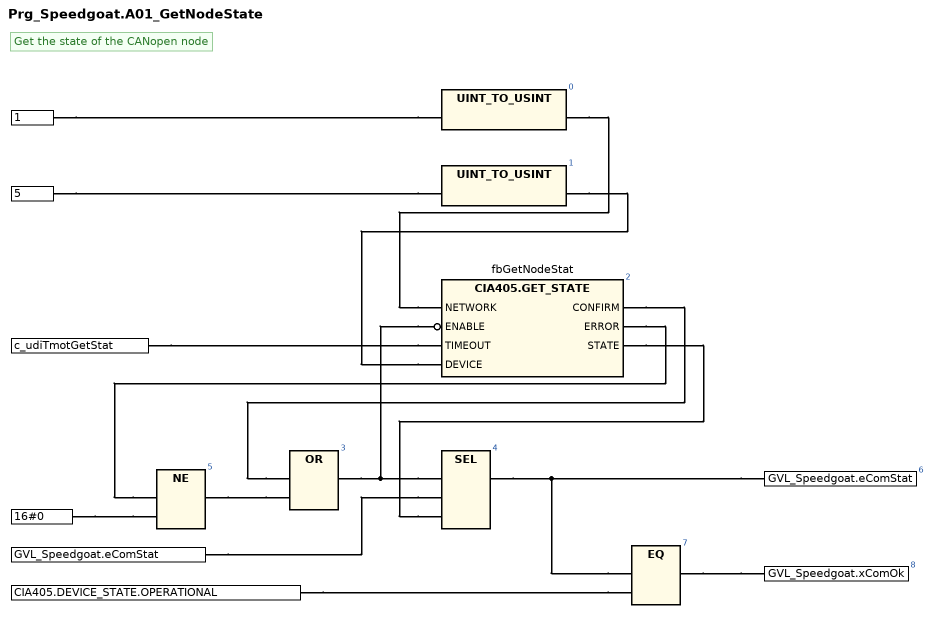
// Get the state of the CANopen node
fbGetNodeStat(
    NETWORK := UINT_TO_USINT(1),
    ENABLE := NOT _w1,
    TIMEOUT := c_udiTmotGetStat,
    DEVICE := UINT_TO_USINT(5)); // CIA405.GET_STATE
_w1 := fbGetNodeStat.CONFIRM OR _w2;
_w3 := SEL(_w1, GVL_Speedgoat.eComStat, fbGetNodeStat.STATE);
_w2 := fbGetNodeStat.ERROR <> 16#0;
GVL_Speedgoat.eComStat := _w3;
GVL_Speedgoat.xComOk := _w3 = CIA405.DEVICE_STATE.OPERATIONAL;
END_ACTION

END_PROGRAM

// HMISAC/Application/AlarmManager
PROGRAM AlarmManager
VAR
END_VAR

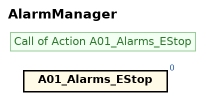
// Call of Action A01_Alarms_EStop
A01_Alarms_EStop();

ACTION A06_Alarms_LXM32i_Node11:
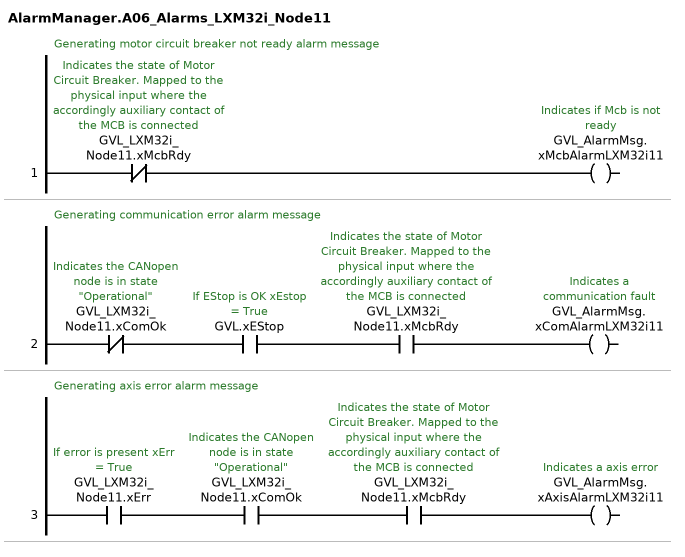
// NETWORK 1
// Generating motor circuit breaker not ready alarm message
//   GVL_LXM32i_Node11.xMcbRdy: Indicates the state of Motor Circuit Breaker. Mapped to the physical input where the accordingly auxiliary contact of the MCB is connected
//   GVL_AlarmMsg.xMcbAlarmLXM32i11: Indicates if Mcb is not ready
GVL_AlarmMsg.xMcbAlarmLXM32i11 := NOT GVL_LXM32i_Node11.xMcbRdy;

// NETWORK 2
// Generating communication error alarm message
//   GVL_LXM32i_Node11.xComOk: Indicates the CANopen node is in state "Operational"
//   GVL.xEStop: If EStop is OK xEstop = True
//   GVL_LXM32i_Node11.xMcbRdy: Indicates the state of Motor Circuit Breaker. Mapped to the physical input where the accordingly auxiliary contact of the MCB is connected
//   GVL_AlarmMsg.xComAlarmLXM32i11: Indicates a communication fault
GVL_AlarmMsg.xComAlarmLXM32i11 := NOT GVL_LXM32i_Node11.xComOk AND GVL.xEStop AND GVL_LXM32i_Node11.xMcbRdy;

// NETWORK 3
// Generating axis error alarm message
//   GVL_LXM32i_Node11.xErr: If error is present xErr = True
//   GVL_LXM32i_Node11.xComOk: Indicates the CANopen node is in state "Operational"
//   GVL_LXM32i_Node11.xMcbRdy: Indicates the state of Motor Circuit Breaker. Mapped to the physical input where the accordingly auxiliary contact of the MCB is connected
//   GVL_AlarmMsg.xAxisAlarmLXM32i11: Indicates a axis error
GVL_AlarmMsg.xAxisAlarmLXM32i11 := GVL_LXM32i_Node11.xErr AND GVL_LXM32i_Node11.xComOk AND GVL_LXM32i_Node11.xMcbRdy;
END_ACTION

ACTION A05_Alarms_LXM28A_Node04:
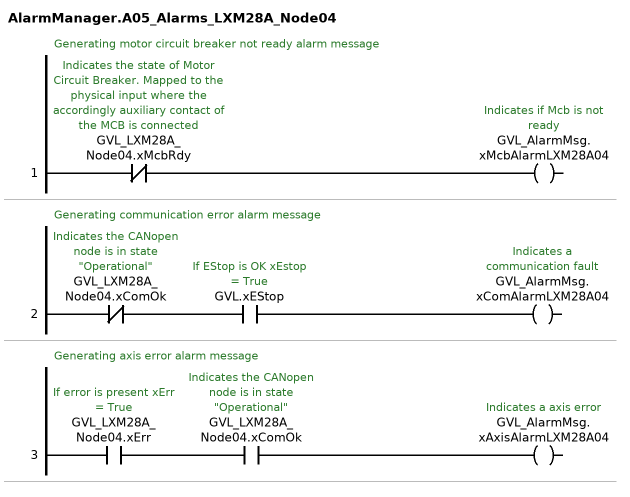
// NETWORK 1
// Generating motor circuit breaker not ready alarm message
//   GVL_LXM28A_Node04.xMcbRdy: Indicates the state of Motor Circuit Breaker. Mapped to the physical input where the accordingly auxiliary contact of the MCB is connected
//   GVL_AlarmMsg.xMcbAlarmLXM28A04: Indicates if Mcb is not ready
GVL_AlarmMsg.xMcbAlarmLXM28A04 := NOT GVL_LXM28A_Node04.xMcbRdy;

// NETWORK 2
// Generating communication error alarm message
//   GVL_LXM28A_Node04.xComOk: Indicates the CANopen node is in state "Operational"
//   GVL.xEStop: If EStop is OK xEstop = True
//   GVL_AlarmMsg.xComAlarmLXM28A04: Indicates a communication fault
GVL_AlarmMsg.xComAlarmLXM28A04 := NOT GVL_LXM28A_Node04.xComOk AND GVL.xEStop;

// NETWORK 3
// Generating axis error alarm message
//   GVL_LXM28A_Node04.xErr: If error is present xErr = True
//   GVL_LXM28A_Node04.xComOk: Indicates the CANopen node is in state "Operational"
//   GVL_AlarmMsg.xAxisAlarmLXM28A04: Indicates a axis error
GVL_AlarmMsg.xAxisAlarmLXM28A04 := GVL_LXM28A_Node04.xErr AND GVL_LXM28A_Node04.xComOk;
END_ACTION

ACTION A01_Alarms_EStop:
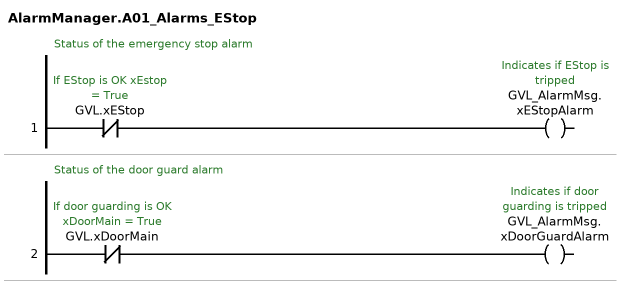
// NETWORK 1
// Status of the emergency stop alarm
//   GVL.xEStop: If EStop is OK xEstop = True
//   GVL_AlarmMsg.xEStopAlarm: Indicates if EStop is tripped
GVL_AlarmMsg.xEStopAlarm := NOT GVL.xEStop;

// NETWORK 2
// Status of the door guard alarm
//   GVL.xDoorMain: If door guarding is OK xDoorMain = True
//   GVL_AlarmMsg.xDoorGuardAlarm: Indicates if door guarding is tripped
GVL_AlarmMsg.xDoorGuardAlarm := NOT GVL.xDoorMain;
END_ACTION

ACTION A04_Alarms_LXM28A_Node03:
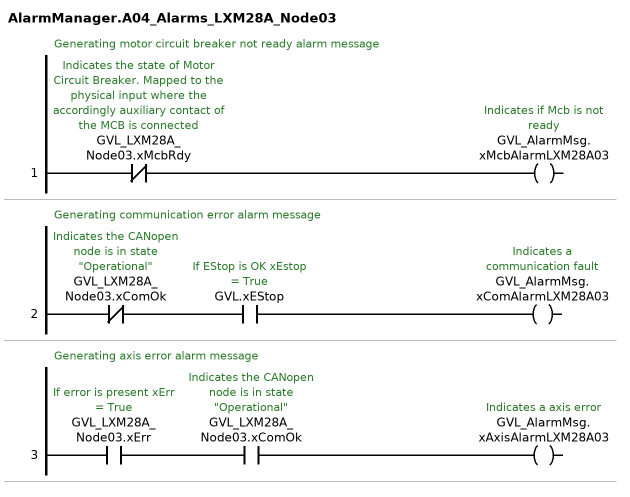
// NETWORK 1
// Generating motor circuit breaker not ready alarm message
//   GVL_LXM28A_Node03.xMcbRdy: Indicates the state of Motor Circuit Breaker. Mapped to the physical input where the accordingly auxiliary contact of the MCB is connected
//   GVL_AlarmMsg.xMcbAlarmLXM28A03: Indicates if Mcb is not ready
GVL_AlarmMsg.xMcbAlarmLXM28A03 := NOT GVL_LXM28A_Node03.xMcbRdy;

// NETWORK 2
// Generating communication error alarm message
//   GVL_LXM28A_Node03.xComOk: Indicates the CANopen node is in state "Operational"
//   GVL.xEStop: If EStop is OK xEstop = True
//   GVL_AlarmMsg.xComAlarmLXM28A03: Indicates a communication fault
GVL_AlarmMsg.xComAlarmLXM28A03 := NOT GVL_LXM28A_Node03.xComOk AND GVL.xEStop;

// NETWORK 3
// Generating axis error alarm message
//   GVL_LXM28A_Node03.xErr: If error is present xErr = True
//   GVL_LXM28A_Node03.xComOk: Indicates the CANopen node is in state "Operational"
//   GVL_AlarmMsg.xAxisAlarmLXM28A03: Indicates a axis error
GVL_AlarmMsg.xAxisAlarmLXM28A03 := GVL_LXM28A_Node03.xErr AND GVL_LXM28A_Node03.xComOk;
END_ACTION

END_PROGRAM

// HMISAC/Application/MAIN
PROGRAM MAIN
VAR
	fbiOneSecPulse: UTIL.BLINK; // FB creation of the 1 second pulse (heartbeat HMI)
	fbGetNodeStat: CIA405.GET_STATE; // FB instance to get the state of the CANopen node	
	fbGrenButnFwdTrigOn: R_TRIG; // FB instance linked to the green forward Butn
	fbGrenButnFwdTrigOff: F_TRIG; // FB instance linked to the green forward Butn
	fbGrenButnRevTrigOn: R_TRIG; // FB instance linked to the green reverse Butn
	fbGrenButnRevTrigOff: F_TRIG; // FB instance linked to the green reverse Butn
	fbRedButnStopTrigOn: F_TRIG; // FB instance linked to the red stop Butn
	fbRedButnStopTrigOff: R_TRIG; // FB instance linked to the red stop Butn
END_VAR
VAR CONSTANT
	c_udiTmotGetStat : UDINT := 1000; // Parameter timeout for fbi CAN0state in ms
END_VAR
VAR // added by the converter: edge detectors and wires of the graphical bodies
    _w1, _w2 : ANY;
END_VAR

// Life bit to HMI
fbiOneSecPulse(ENABLE := TRUE, TIMELOW := T#1S, TIMEHIGH := T#1S);
GVL.xPulse_1s := fbiOneSecPulse.OUT;
GVL.xstart :=1;
// Cyclic call of Actions
A01_CANopen_Slave_State();
A02_CANopen_State();
//A04_Device_Error_State();

ACTION A02_CANopen_State:
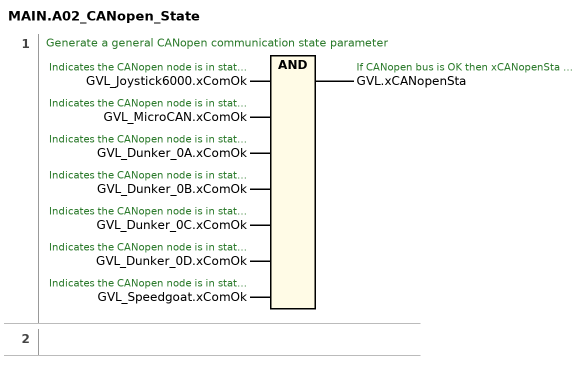
// NETWORK 1
// Generate a general CANopen communication state parameter
//   GVL_Joystick6000.xComOk: Indicates the CANopen node is in state "Operational"
//   GVL_MicroCAN.xComOk: Indicates the CANopen node is in state "Operational"
//   GVL_Dunker_0A.xComOk: Indicates the CANopen node is in state "Operational"
//   GVL_Dunker_0B.xComOk: Indicates the CANopen node is in state "Operational"
//   GVL_Dunker_0C.xComOk: Indicates the CANopen node is in state "Operational"
//   GVL_Dunker_0D.xComOk: Indicates the CANopen node is in state "Operational"
//   GVL_Speedgoat.xComOk: Indicates the CANopen node is in state "Operational"
//   GVL.xCANopenSta: If CANopen bus is OK then xCANopenSta = TRUE
GVL.xCANopenSta := GVL_Joystick6000.xComOk AND GVL_MicroCAN.xComOk AND GVL_Dunker_0A.xComOk AND GVL_Dunker_0B.xComOk AND GVL_Dunker_0C.xComOk AND GVL_Dunker_0D.xComOk AND GVL_Speedgoat.xComOk;

// NETWORK 2
END_ACTION

ACTION A04_Device_Error_State:
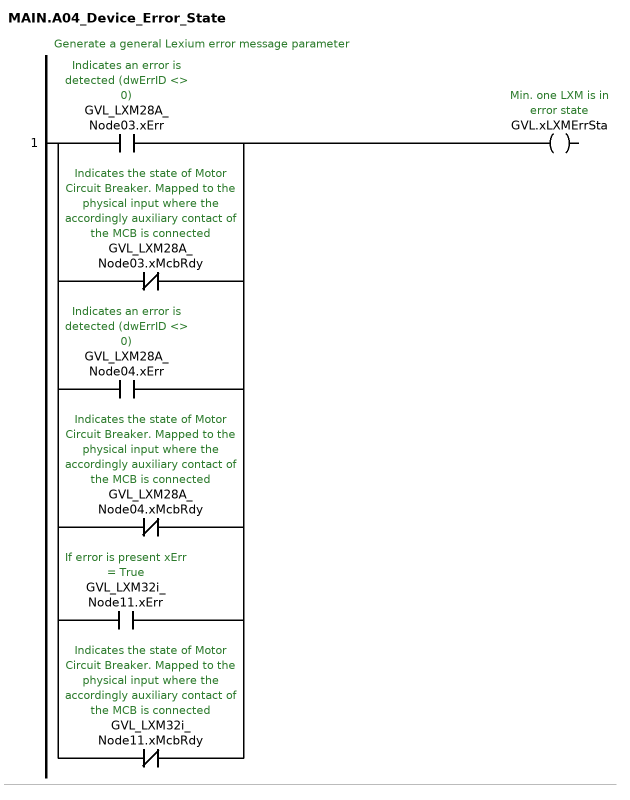
// NETWORK 1
// Generate a general Lexium error message parameter
//   GVL_LXM28A_Node03.xErr: Indicates an error is detected (dwErrID <> 0)
//   GVL_LXM28A_Node03.xMcbRdy: Indicates the state of Motor Circuit Breaker. Mapped to the physical input where the accordingly auxiliary contact of the MCB is connected
//   GVL_LXM28A_Node04.xErr: Indicates an error is detected (dwErrID <> 0)
//   GVL_LXM28A_Node04.xMcbRdy: Indicates the state of Motor Circuit Breaker. Mapped to the physical input where the accordingly auxiliary contact of the MCB is connected
//   GVL_LXM32i_Node11.xErr: If error is present xErr = True
//   GVL_LXM32i_Node11.xMcbRdy: Indicates the state of Motor Circuit Breaker. Mapped to the physical input where the accordingly auxiliary contact of the MCB is connected
//   GVL.xLXMErrSta: Min. one LXM is in error state
GVL.xLXMErrSta := GVL_LXM28A_Node03.xErr OR NOT GVL_LXM28A_Node03.xMcbRdy OR GVL_LXM28A_Node04.xErr OR NOT GVL_LXM28A_Node04.xMcbRdy OR GVL_LXM32i_Node11.xErr OR NOT GVL_LXM32i_Node11.xMcbRdy;
END_ACTION

ACTION A01_CANopen_Slave_State:
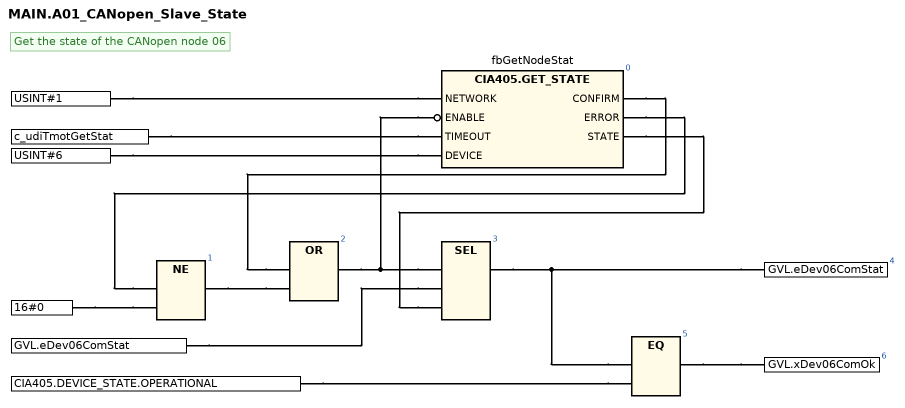
// Get the state of the CANopen node 06
fbGetNodeStat(NETWORK := USINT#1, ENABLE := NOT _w1, TIMEOUT := c_udiTmotGetStat, DEVICE := USINT#6); // CIA405.GET_STATE
_w1 := fbGetNodeStat.CONFIRM OR fbGetNodeStat.ERROR <> 16#0;
_w2 := SEL(_w1, GVL.eDev06ComStat, fbGetNodeStat.STATE);
GVL.eDev06ComStat := _w2;
GVL.xDev06ComOk := _w2 = CIA405.DEVICE_STATE.OPERATIONAL;
END_ACTION

END_PROGRAM

// HMISAC/Application/OutputMapping
PROGRAM OutputMapping
VAR
END_VAR

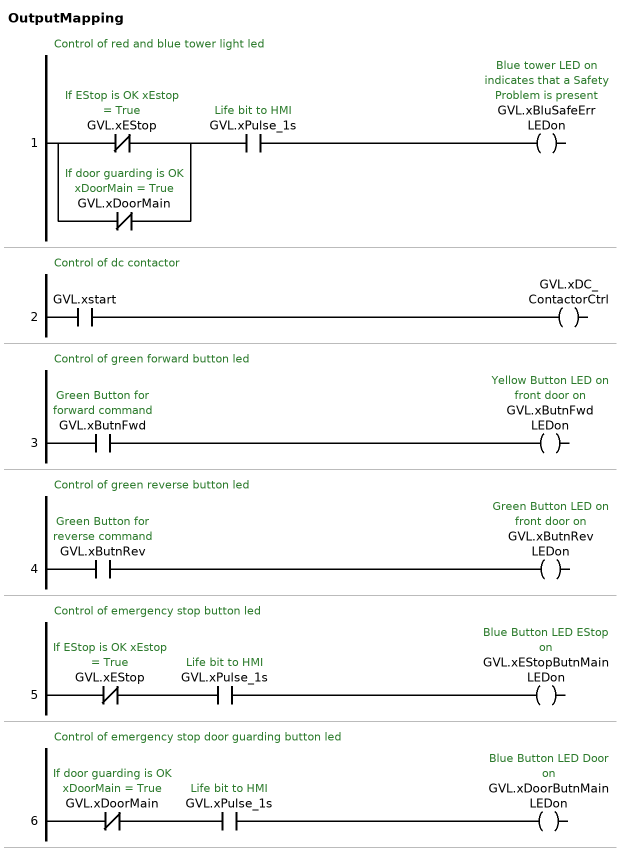
// NETWORK 1
// Control of red and blue tower light led
//   GVL.xEStop: If EStop is OK xEstop = True
//   GVL.xDoorMain: If door guarding is OK xDoorMain = True
//   GVL.xPulse_1s: Life bit to HMI
//   GVL.xBluSafeErrLEDon: Blue tower LED on indicates that a Safety Problem is present
GVL.xBluSafeErrLEDon := (NOT GVL.xEStop OR NOT GVL.xDoorMain) AND GVL.xPulse_1s;

// NETWORK 2
// Control of dc contactor
GVL.xDC_ContactorCtrl := GVL.xstart;

// NETWORK 3
// Control of green forward button led
//   GVL.xButnFwd: Green Button for forward command
//   GVL.xButnFwdLEDon: Yellow Button LED on front door on
GVL.xButnFwdLEDon := GVL.xButnFwd;

// NETWORK 4
// Control of green reverse button led
//   GVL.xButnRev: Green Button for reverse command
//   GVL.xButnRevLEDon: Green Button LED on front door on
GVL.xButnRevLEDon := GVL.xButnRev;

// NETWORK 5
// Control of emergency stop button led
//   GVL.xEStop: If EStop is OK xEstop = True
//   GVL.xPulse_1s: Life bit to HMI
//   GVL.xEStopButnMainLEDon: Blue Button LED EStop on
GVL.xEStopButnMainLEDon := NOT GVL.xEStop AND GVL.xPulse_1s;

// NETWORK 6
// Control of emergency stop door guarding button led
//   GVL.xDoorMain: If door guarding is OK xDoorMain = True
//   GVL.xPulse_1s: Life bit to HMI
//   GVL.xDoorButnMainLEDon: Blue Button LED Door on
GVL.xDoorButnMainLEDon := NOT GVL.xDoorMain AND GVL.xPulse_1s;

END_PROGRAM

// HMISAC/Application/Prg_WriteParameter
PROGRAM Prg_WriteParameter
VAR
	fbWriteParaLXM2803	:SEM_LXM28.MC_WriteParameter_LXM28; // FB instance to write parameter (CANopen objects) to the LXM28 drive
	fbWriteParaLXM2804	:SEM_LXM28.MC_WriteParameter_LXM28; // FB instance to write parameter (CANopen objects) to the LXM28 drive
	
	byStatWriteParaLXM2803	:BYTE;	// Status parameter write procedure, Bit 0 = 0x6083 is written, Bit 1 = 0x6083 is written, ...
	byStatWriteParaLXM2804	:BYTE;	// Status parameter write procedure, Bit 0 = 0x6083 is written, Bit 1 = 0x6083 is written, ...
	
	byAlarmWriteParaLXM2803	:BYTE;	// Status parameter write procedure, Bit 0 = 0x6083 is written, Bit 1 = 0x6083 is written, ...
	byAlarmWriteParaLXM2804	:BYTE;	// Error ocurred during parameter write procedure, Bit 0 = 0x6083, Bit 1 = 0x6083, ...
	
	uiStatWriteParaLXM2803	:UINT;	// aux variable for case instruction
	uiStatWriteParaLXM2804	:UINT;	// aux variable for case instruction
	
	xAutoInitLXM2803	:BOOL:=TRUE;	// TRUE means the parameter will be written on each (re)start of the CAN communication
	xAutoInitLXM2804	:BOOL:=TRUE;	// TRUE means the parameter will be written on each (re)start of the CAN communication
	
	udiOldValParaAccLXM2803		:UDINT;	// old value of the parameter which was successfully written
	udiOldValParaDecLXM2803		:UDINT;	// old value of the parameter which was successfully written
	udiOldValParaDecStopLXM2803	:UDINT;	// old value of the parameter which was successfully written
	udiOldValParaAccLXM2804		:UDINT;	// old value of the parameter which was successfully written
	udiOldValParaDecLXM2804		:UDINT;	// old value of the parameter which was successfully written
	udiOldValParaDecStopLXM2804	:UDINT;	// old value of the parameter which was successfully written
END_VAR
VAR CONSTANT
END_VAR

//A_WriteParameter_LXM2803();
//A_WriteParameter_LXM2804();

ACTION A_WriteParameter_LXM2804:
(*Reset status when communication is down*)
IF NOT GVL_LXM28A_Node04.xComOk THEN
	byStatWriteParaLXM2804	:= 0;
	xAutoInitLXM2804		:= TRUE;	// after communication restart the parameters will be written again 
END_IF

CASE uiStatWriteParaLXM2804 OF
	0:	(*wait for request*)
		IF GVL_LXM28A_Node04.xComOk AND NOT GVL_LXM28A_Node04.xErr THEN
			IF GVL_HmiVar.xCmdWriteParaLXM28A04 THEN
				byStatWriteParaLXM2804				:= 0;
				uiStatWriteParaLXM2804				:= 10;
				GVL_HmiVar.xCmdWriteParaLXM28A04	:= FALSE;
			ELSIF xAutoInitLXM2804 AND (byStatWriteParaLXM2804 <> 7) THEN
				IF NOT byStatWriteParaLXM2804.0 THEN
					uiStatWriteParaLXM2804	:= 10;
				ELSIF NOT byStatWriteParaLXM2804.1 THEN
					uiStatWriteParaLXM2804	:= 20;
				ELSIF NOT byStatWriteParaLXM2804.2 THEN
					uiStatWriteParaLXM2804	:= 30;	
				END_IF
			END_IF
		END_IF
	10:	(*Write parameter 0x6083*)
		fbWriteParaLXM2804.Execute			:= TRUE;
		fbWriteParaLXM2804.ParameterNumber	:= 1000;
		fbWriteParaLXM2804.Index			:= 16#6083;
		fbWriteParaLXM2804.Length			:= 4;
		fbWriteParaLXM2804.Value			:= UDINT_TO_DINT(GVL_Retain.udiParaAccLXM2804);
		IF fbWriteParaLXM2804.Done OR fbWriteParaLXM2804.Error THEN
			fbWriteParaLXM2804.Execute	:= FALSE;
			IF fbWriteParaLXM2804.Done THEN
				byStatWriteParaLXM2804.0 	:= fbWriteParaLXM2804.Done;
				udiOldValParaAccLXM2804		:= DINT_TO_UDINT(fbWriteParaLXM2804.Value);	// store the written value
			END_IF
			byAlarmWriteParaLXM2804.0	:= fbWriteParaLXM2804.Error;
			uiStatWriteParaLXM2804		:= 20;
		END_IF
	20:	(*Write parameter 0x6084*)
		fbWriteParaLXM2804.Execute			:= TRUE;
		fbWriteParaLXM2804.ParameterNumber	:= 1000;
		fbWriteParaLXM2804.Index			:= 16#6084;
		fbWriteParaLXM2804.Length			:= 4;
		fbWriteParaLXM2804.Value			:= UDINT_TO_DINT(GVL_Retain.udiParaDecLXM2804);
		IF fbWriteParaLXM2804.Done OR fbWriteParaLXM2804.Error THEN
			fbWriteParaLXM2804.Execute	:= FALSE;
			IF fbWriteParaLXM2804.Done THEN
				byStatWriteParaLXM2804.1 	:= fbWriteParaLXM2804.Done;
				udiOldValParaDecLXM2804		:= DINT_TO_UDINT(fbWriteParaLXM2804.Value);	// store the written value
			END_IF
			byAlarmWriteParaLXM2804.1	:= fbWriteParaLXM2804.Error;
			uiStatWriteParaLXM2804		:= 30;
		END_IF
	30:	(*Write parameter 0x6085*)
		fbWriteParaLXM2804.Execute			:= TRUE;
		fbWriteParaLXM2804.ParameterNumber	:= 1000;
		fbWriteParaLXM2804.Index			:= 16#6085;
		fbWriteParaLXM2804.Length			:= 4;
		fbWriteParaLXM2804.Value			:= UDINT_TO_DINT(GVL_Retain.udiParaDecStopLXM2804);
		IF fbWriteParaLXM2804.Done OR fbWriteParaLXM2804.Error THEN
			fbWriteParaLXM2804.Execute	:= FALSE;
			IF fbWriteParaLXM2804.Done THEN
				byStatWriteParaLXM2804.2 		:= fbWriteParaLXM2804.Done;
				udiOldValParaDecStopLXM2804		:= DINT_TO_UDINT(fbWriteParaLXM2804.Value);	// store the written value
			END_IF
			byAlarmWriteParaLXM2804.2	:= fbWriteParaLXM2804.Error;
			uiStatWriteParaLXM2804		:= 0;
		END_IF	
END_CASE
(*Call of the Function Block*)
fbWriteParaLXM2804(Axis:=LXM28A_Node04);

(*Reset AutoInit if all parameters have been written succesfully*)
xAutoInitLXM2804	R= (byStatWriteParaLXM2804 = 7);

(*Check if value on HMI has changed and reset the "done" flag* if so*)
byStatWriteParaLXM2804.0	R= udiOldValParaAccLXM2804 <> GVL_Retain.udiParaAccLXM2804;
byStatWriteParaLXM2804.1	R= udiOldValParaDecLXM2804 <> GVL_Retain.udiParaDecLXM2804;
byStatWriteParaLXM2804.2	R= udiOldValParaDecStopLXM2804 <> GVL_Retain.udiParaDecStopLXM2804;

(*update status variables for HMI*)
GVL_HmiVar.xWriteParaAccDoneLXM2804		:=byStatWriteParaLXM2804.0;
GVL_HmiVar.xWriteParaDecDoneLXM2804		:=byStatWriteParaLXM2804.1;
GVL_HmiVar.xWriteParaDecStopDoneLXM2804	:=byStatWriteParaLXM2804.2;
(*Generate Alarm if write parameter have been failed*)
GVL_AlarmMsg.xAlrmWriteParaLXM28A04		:=(byAlarmWriteParaLXM2804 <> 0);
END_ACTION

ACTION A_WriteParameter_LXM2803:
(*Reset status when communication is down*)
IF NOT GVL_LXM28A_Node03.xComOk THEN
	byStatWriteParaLXM2803	:= 0;
	xAutoInitLXM2803		:= TRUE;	// after communication restart the parameters will be written again 
END_IF

CASE uiStatWriteParaLXM2803 OF
	0:	(*wait for request*)
		IF GVL_LXM28A_Node03.xComOk AND NOT GVL_LXM28A_Node03.xErr THEN
			IF GVL_HmiVar.xCmdWriteParaLXM28A03 THEN
				byStatWriteParaLXM2803				:= 0;
				uiStatWriteParaLXM2803				:= 10;
				GVL_HmiVar.xCmdWriteParaLXM28A03	:= FALSE;
			ELSIF xAutoInitLXM2803 AND (byStatWriteParaLXM2803 <> 7) THEN
				IF NOT byStatWriteParaLXM2803.0 THEN
					uiStatWriteParaLXM2803	:= 10;
				ELSIF NOT byStatWriteParaLXM2803.1 THEN
					uiStatWriteParaLXM2803	:= 20;
				ELSIF NOT byStatWriteParaLXM2803.2 THEN
					uiStatWriteParaLXM2803	:= 30;	
				END_IF
			END_IF
		END_IF
	10:	(*Write parameter 0x6083*)
		fbWriteParaLXM2803.Execute			:= TRUE;
		fbWriteParaLXM2803.ParameterNumber	:= 1000;
		fbWriteParaLXM2803.Index			:= 16#6083;
		fbWriteParaLXM2803.Length			:= 4;
		fbWriteParaLXM2803.Value			:= UDINT_TO_DINT(GVL_Retain.udiParaAccLXM2803);
		IF fbWriteParaLXM2803.Done OR fbWriteParaLXM2803.Error THEN
			fbWriteParaLXM2803.Execute	:= FALSE;
			IF fbWriteParaLXM2803.Done THEN
				byStatWriteParaLXM2803.0 	:= fbWriteParaLXM2803.Done;
				udiOldValParaAccLXM2803		:= DINT_TO_UDINT(fbWriteParaLXM2803.Value);	// store the written value
			END_IF
			byAlarmWriteParaLXM2803.0	:= fbWriteParaLXM2803.Error;
			uiStatWriteParaLXM2803		:= 20;
		END_IF
	20:	(*Write parameter 0x6084*)
		fbWriteParaLXM2803.Execute			:= TRUE;
		fbWriteParaLXM2803.ParameterNumber	:= 1000;
		fbWriteParaLXM2803.Index			:= 16#6084;
		fbWriteParaLXM2803.Length			:= 4;
		fbWriteParaLXM2803.Value			:= UDINT_TO_DINT(GVL_Retain.udiParaDecLXM2803);
		IF fbWriteParaLXM2803.Done OR fbWriteParaLXM2803.Error THEN
			fbWriteParaLXM2803.Execute	:= FALSE;
			IF fbWriteParaLXM2803.Done THEN
				byStatWriteParaLXM2803.1 	:= fbWriteParaLXM2803.Done;
				udiOldValParaDecLXM2803		:= DINT_TO_UDINT(fbWriteParaLXM2803.Value);	// store the written value
			END_IF
			byAlarmWriteParaLXM2803.1	:= fbWriteParaLXM2803.Error;
			uiStatWriteParaLXM2803		:= 30;
		END_IF
	30:	(*Write parameter 0x6085*)
		fbWriteParaLXM2803.Execute			:= TRUE;
		fbWriteParaLXM2803.ParameterNumber	:= 1000;
		fbWriteParaLXM2803.Index			:= 16#6085;
		fbWriteParaLXM2803.Length			:= 4;
		fbWriteParaLXM2803.Value			:= UDINT_TO_DINT(GVL_Retain.udiParaDecStopLXM2803);
		IF fbWriteParaLXM2803.Done OR fbWriteParaLXM2803.Error THEN
			fbWriteParaLXM2803.Execute	:= FALSE;
			IF fbWriteParaLXM2803.Done THEN
				byStatWriteParaLXM2803.2 		:= fbWriteParaLXM2803.Done;
				udiOldValParaDecStopLXM2803		:= DINT_TO_UDINT(fbWriteParaLXM2803.Value);	// store the written value
			END_IF
			byAlarmWriteParaLXM2803.2	:= fbWriteParaLXM2803.Error;
			uiStatWriteParaLXM2803		:= 0;
		END_IF	
END_CASE
(*Call of the Function Block*)
fbWriteParaLXM2803(Axis:=LXM28A_Node03);

(*Reset AutoInit if all parameters have been written succesfully*)
xAutoInitLXM2803	R= (byStatWriteParaLXM2803 = 7);

(*Check if value on HMI has changed and reset the "done" flag* if so*)
byStatWriteParaLXM2803.0	R= udiOldValParaAccLXM2803 <> GVL_Retain.udiParaAccLXM2803;
byStatWriteParaLXM2803.1	R= udiOldValParaDecLXM2803 <> GVL_Retain.udiParaDecLXM2803;
byStatWriteParaLXM2803.2	R= udiOldValParaDecStopLXM2803 <> GVL_Retain.udiParaDecStopLXM2803;

(*update status variables for HMI*)
GVL_HmiVar.xWriteParaAccDoneLXM2803		:=byStatWriteParaLXM2803.0;
GVL_HmiVar.xWriteParaDecDoneLXM2803		:=byStatWriteParaLXM2803.1;
GVL_HmiVar.xWriteParaDecStopDoneLXM2803	:=byStatWriteParaLXM2803.2;
(*Generate Alarm if write parameter have been failed*)
GVL_AlarmMsg.xAlrmWriteParaLXM28A03		:=(byAlarmWriteParaLXM2803 <> 0);
END_ACTION

END_PROGRAM

// HMISAC/Application/LXM32i_Node11/Prg_LXM32i_Node11
PROGRAM Prg_LXM32i_Node11
VAR
	fbGetNodeStat     : CIA405.GET_STATE; // FB instance to get the state of the CANopen node
	fbPwrLXM		  : SEM_LXM32i.MC_Power_LXM32i; // FB instance to power the Lexium
	fbRstLXM		  : SEM_LXM32i.MC_Reset_LXM32i; // FB instance to reset the Lexium
	fbStopLXM		  : SEM_LXM32i.MC_Stop_LXM32i; // FB instance to stop the Lexium
	fbJogLXM		  : SEM_LXM32i.MC_Jog_LXM32i; // FB instance to turn the drive manually
	fbVeloLXM	 	  : SEM_LXM32i.MC_MoveVelocity_LXM32i; // FB instance to start the Lexium in operating mode Profile Velocity
	fbRelLXM	 	  : SEM_LXM32i.MC_MoveRelative_LXM32i; // FB instance to start a movement by the defined distance
	fbAbsLXM	 	  : SEM_LXM32i.MC_MoveAbsolute_LXM32i; // FB instance to start a movement to the defined absolute target position
	fbErrLXM	 	  : SEM_LXM32i.MC_ReadAxisError_LXM32i; // FB instance to read the error state of the Lexium
	fbHomeLXM	  	  : SEM_LXM32i.MC_Home_LXM32i; // FB instance to start a reference movement					
END_VAR
VAR CONSTANT
	c_udiTmotGetStat : UDINT := 1000; // Parameter timeout for FB GET_STATE in ms
END_VAR
VAR // added by the converter: edge detectors and wires of the graphical bodies
    _w1, _w2 : ANY;
END_VAR

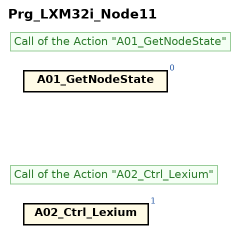
// Call of the Action "A01_GetNodeState"
A01_GetNodeState();
// Call of the Action "A02_Ctrl_Lexium"
A02_Ctrl_Lexium();

ACTION A02_Ctrl_Lexium:
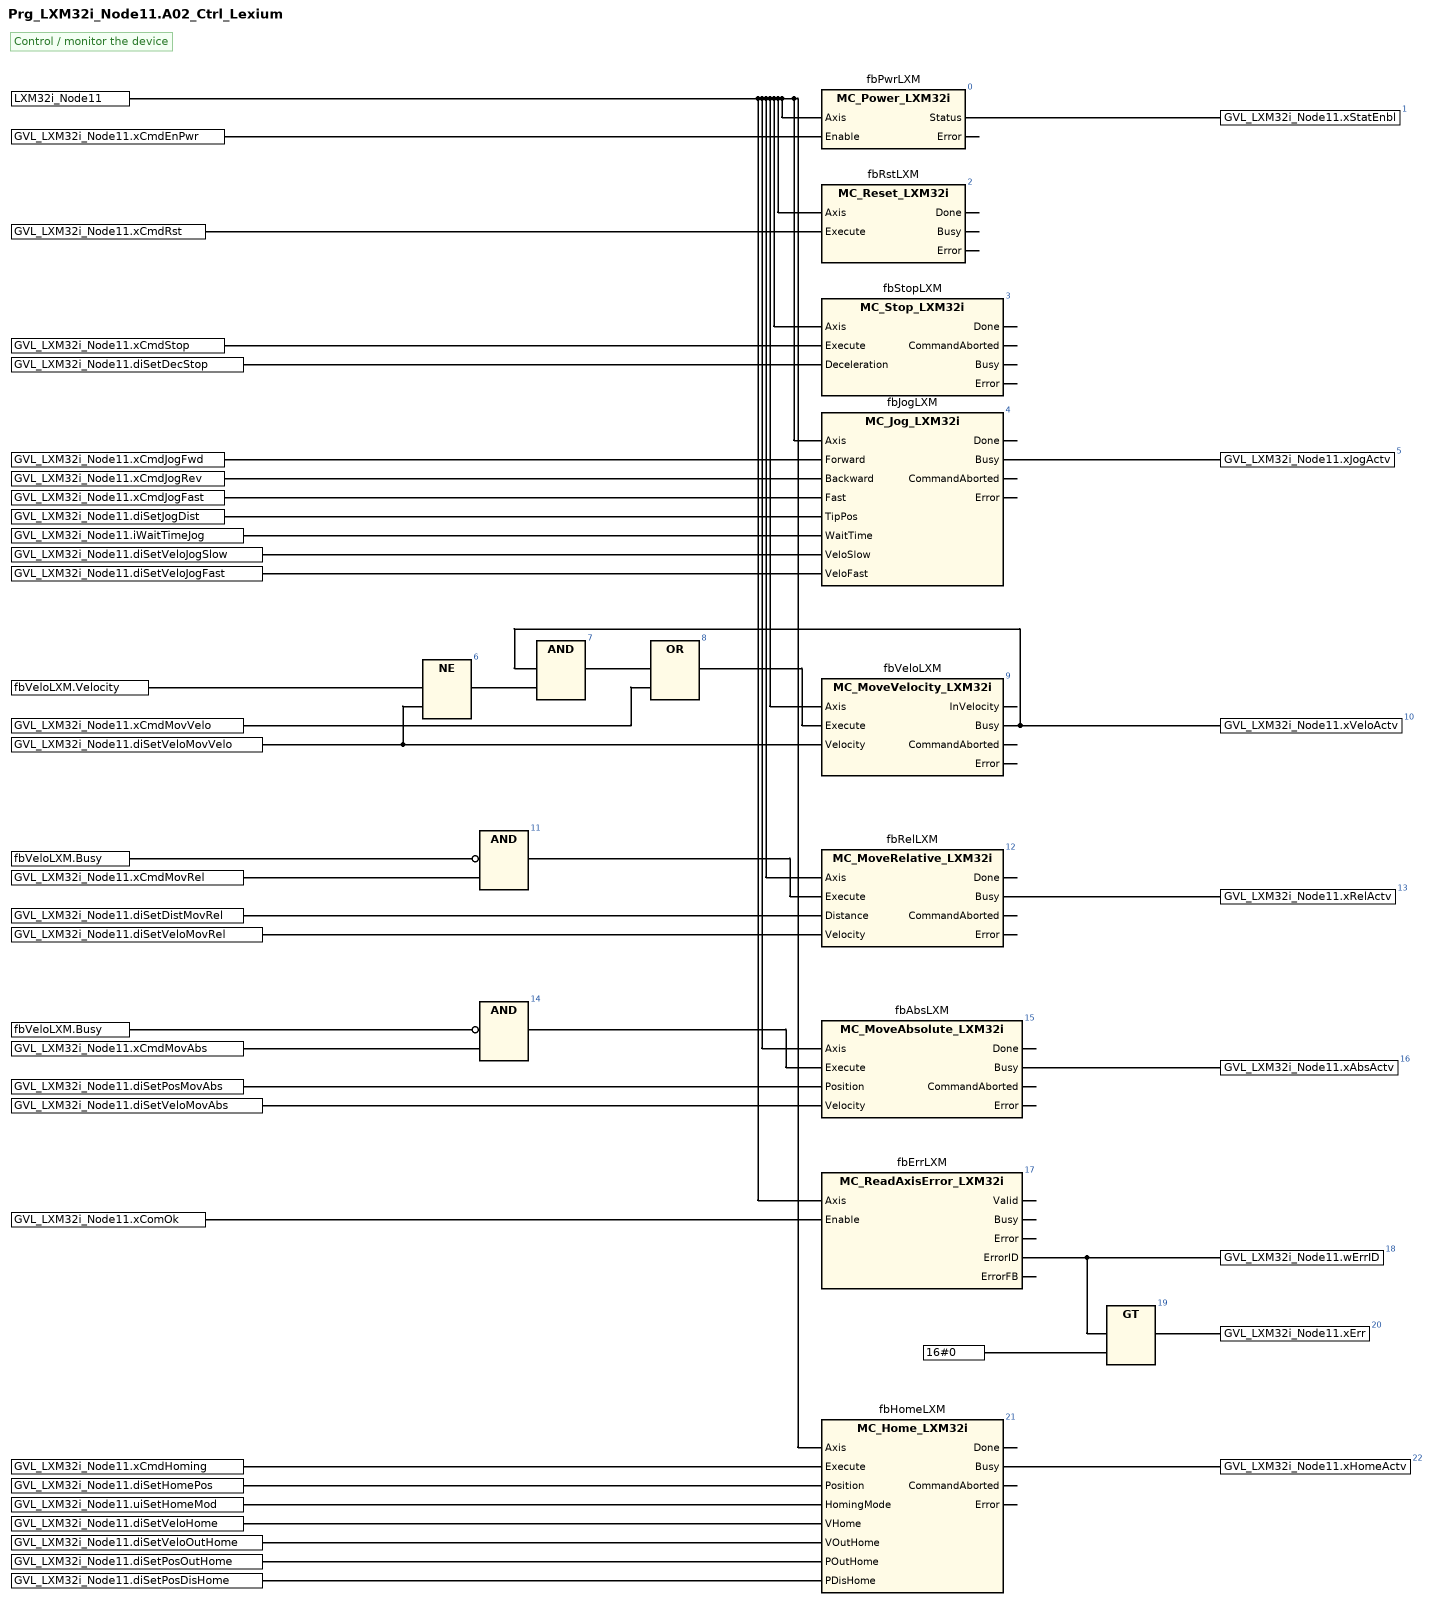
// Control / monitor the device
fbPwrLXM(Axis := LXM32i_Node11, Enable := GVL_LXM32i_Node11.xCmdEnPwr); // MC_Power_LXM32i
GVL_LXM32i_Node11.xStatEnbl := fbPwrLXM.Status;
fbRstLXM(Axis := LXM32i_Node11, Execute := GVL_LXM32i_Node11.xCmdRst); // MC_Reset_LXM32i
fbStopLXM(
    Axis := LXM32i_Node11,
    Execute := GVL_LXM32i_Node11.xCmdStop,
    Deceleration := GVL_LXM32i_Node11.diSetDecStop); // MC_Stop_LXM32i
fbJogLXM(
    Axis := LXM32i_Node11,
    Forward := GVL_LXM32i_Node11.xCmdJogFwd,
    Backward := GVL_LXM32i_Node11.xCmdJogRev,
    Fast := GVL_LXM32i_Node11.xCmdJogFast,
    TipPos := GVL_LXM32i_Node11.diSetJogDist,
    WaitTime := GVL_LXM32i_Node11.iWaitTimeJog,
    VeloSlow := GVL_LXM32i_Node11.diSetVeloJogSlow,
    VeloFast := GVL_LXM32i_Node11.diSetVeloJogFast); // MC_Jog_LXM32i
GVL_LXM32i_Node11.xJogActv := fbJogLXM.Busy;
fbVeloLXM(
    Axis := LXM32i_Node11,
    Execute := fbVeloLXM.Busy AND fbVeloLXM.Velocity <> GVL_LXM32i_Node11.diSetVeloMovVelo OR GVL_LXM32i_Node11.xCmdMovVelo,
    Velocity := GVL_LXM32i_Node11.diSetVeloMovVelo); // MC_MoveVelocity_LXM32i
GVL_LXM32i_Node11.xVeloActv := fbVeloLXM.Busy;
fbRelLXM(
    Axis := LXM32i_Node11,
    Execute := NOT fbVeloLXM.Busy AND GVL_LXM32i_Node11.xCmdMovRel,
    Distance := GVL_LXM32i_Node11.diSetDistMovRel,
    Velocity := GVL_LXM32i_Node11.diSetVeloMovRel); // MC_MoveRelative_LXM32i
GVL_LXM32i_Node11.xRelActv := fbRelLXM.Busy;
fbAbsLXM(
    Axis := LXM32i_Node11,
    Execute := NOT fbVeloLXM.Busy AND GVL_LXM32i_Node11.xCmdMovAbs,
    Position := GVL_LXM32i_Node11.diSetPosMovAbs,
    Velocity := GVL_LXM32i_Node11.diSetVeloMovAbs); // MC_MoveAbsolute_LXM32i
GVL_LXM32i_Node11.xAbsActv := fbAbsLXM.Busy;
fbErrLXM(Axis := LXM32i_Node11, Enable := GVL_LXM32i_Node11.xComOk); // MC_ReadAxisError_LXM32i
GVL_LXM32i_Node11.wErrID := fbErrLXM.ErrorID;
GVL_LXM32i_Node11.xErr := fbErrLXM.ErrorID > 16#0;
fbHomeLXM(
    Axis := LXM32i_Node11,
    Execute := GVL_LXM32i_Node11.xCmdHoming,
    Position := GVL_LXM32i_Node11.diSetHomePos,
    HomingMode := GVL_LXM32i_Node11.uiSetHomeMod,
    VHome := GVL_LXM32i_Node11.diSetVeloHome,
    VOutHome := GVL_LXM32i_Node11.diSetVeloOutHome,
    POutHome := GVL_LXM32i_Node11.diSetPosOutHome,
    PDisHome := GVL_LXM32i_Node11.diSetPosDisHome); // MC_Home_LXM32i
GVL_LXM32i_Node11.xHomeActv := fbHomeLXM.Busy;
END_ACTION

ACTION A01_GetNodeState:
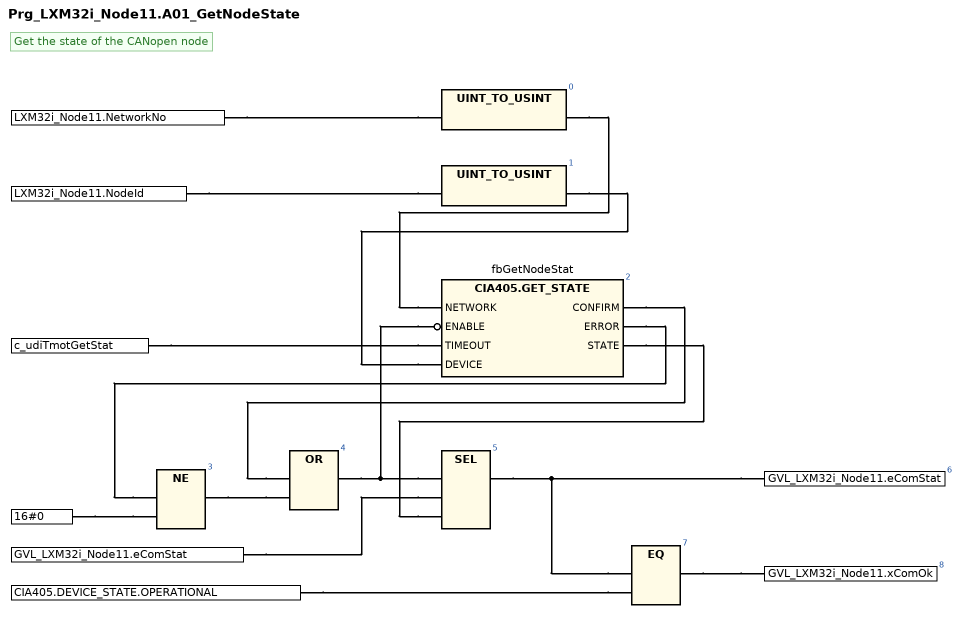
// Get the state of the CANopen node
fbGetNodeStat(
    NETWORK := UINT_TO_USINT(LXM32i_Node11.NetworkNo),
    ENABLE := NOT _w1,
    TIMEOUT := c_udiTmotGetStat,
    DEVICE := UINT_TO_USINT(LXM32i_Node11.NodeId)); // CIA405.GET_STATE
_w1 := fbGetNodeStat.CONFIRM OR fbGetNodeStat.ERROR <> 16#0;
_w2 := SEL(_w1, GVL_LXM32i_Node11.eComStat, fbGetNodeStat.STATE);
GVL_LXM32i_Node11.eComStat := _w2;
GVL_LXM32i_Node11.xComOk := _w2 = CIA405.DEVICE_STATE.OPERATIONAL;
END_ACTION

END_PROGRAM

// HMISAC/Application/LXM28A_Node03/Prg_LXM28A_Node03
PROGRAM Prg_LXM28A_Node03
VAR
	fbGetNodeStat     : CIA405.GET_STATE; // FB instance to get the state of the CANopen node
	fbPwrLXM28		  : SEM_LXM28.MC_Power_LXM28; // FB instance to power the Lexium
	fbRstLXM28		  : SEM_LXM28.MC_Reset_LXM28; // FB instance to reset the Lexium
	fbStopLXM28		  : SEM_LXM28.MC_Stop_LXM28; // FB instance to stop the Lexium
	fbJogLXM28		  : SEM_LXM28.MC_Jog_LXM28; // FB instance to turn the drive manually
	fbVeloLXM28	 	  : SEM_LXM28.MC_MoveVelocity_LXM28; // FB instance to start the Lexium in operating mode Profile Velocity
	fbRelLXM28	 	  : SEM_LXM28.MC_MoveRelative_LXM28; // FB instance to start a movement by the defined distance
	fbAbsLXM28	 	  : SEM_LXM28.MC_MoveAbsolute_LXM28; // FB instance to start a movement to the defined absolute target position
	fbErrLXM28	 	  : SEM_LXM28.MC_ReadAxisError_LXM28; // FB instance to read the error state of the Lexium
	fbHomeLXM28	  	  : SEM_LXM28.MC_Home_LXM28; // FB instance to start a reference movement					
END_VAR
VAR CONSTANT
	c_udiTmotGetStat : UDINT := 1000; // Parameter timeout for FB GET_STATE in ms
END_VAR
VAR // added by the converter: edge detectors and wires of the graphical bodies
    _w1, _w2 : ANY;
END_VAR

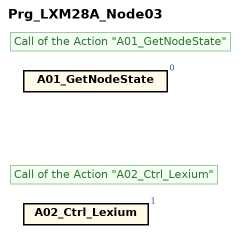
// Call of the Action "A01_GetNodeState"
A01_GetNodeState();
// Call of the Action "A02_Ctrl_Lexium"
A02_Ctrl_Lexium();

ACTION A02_Ctrl_Lexium:
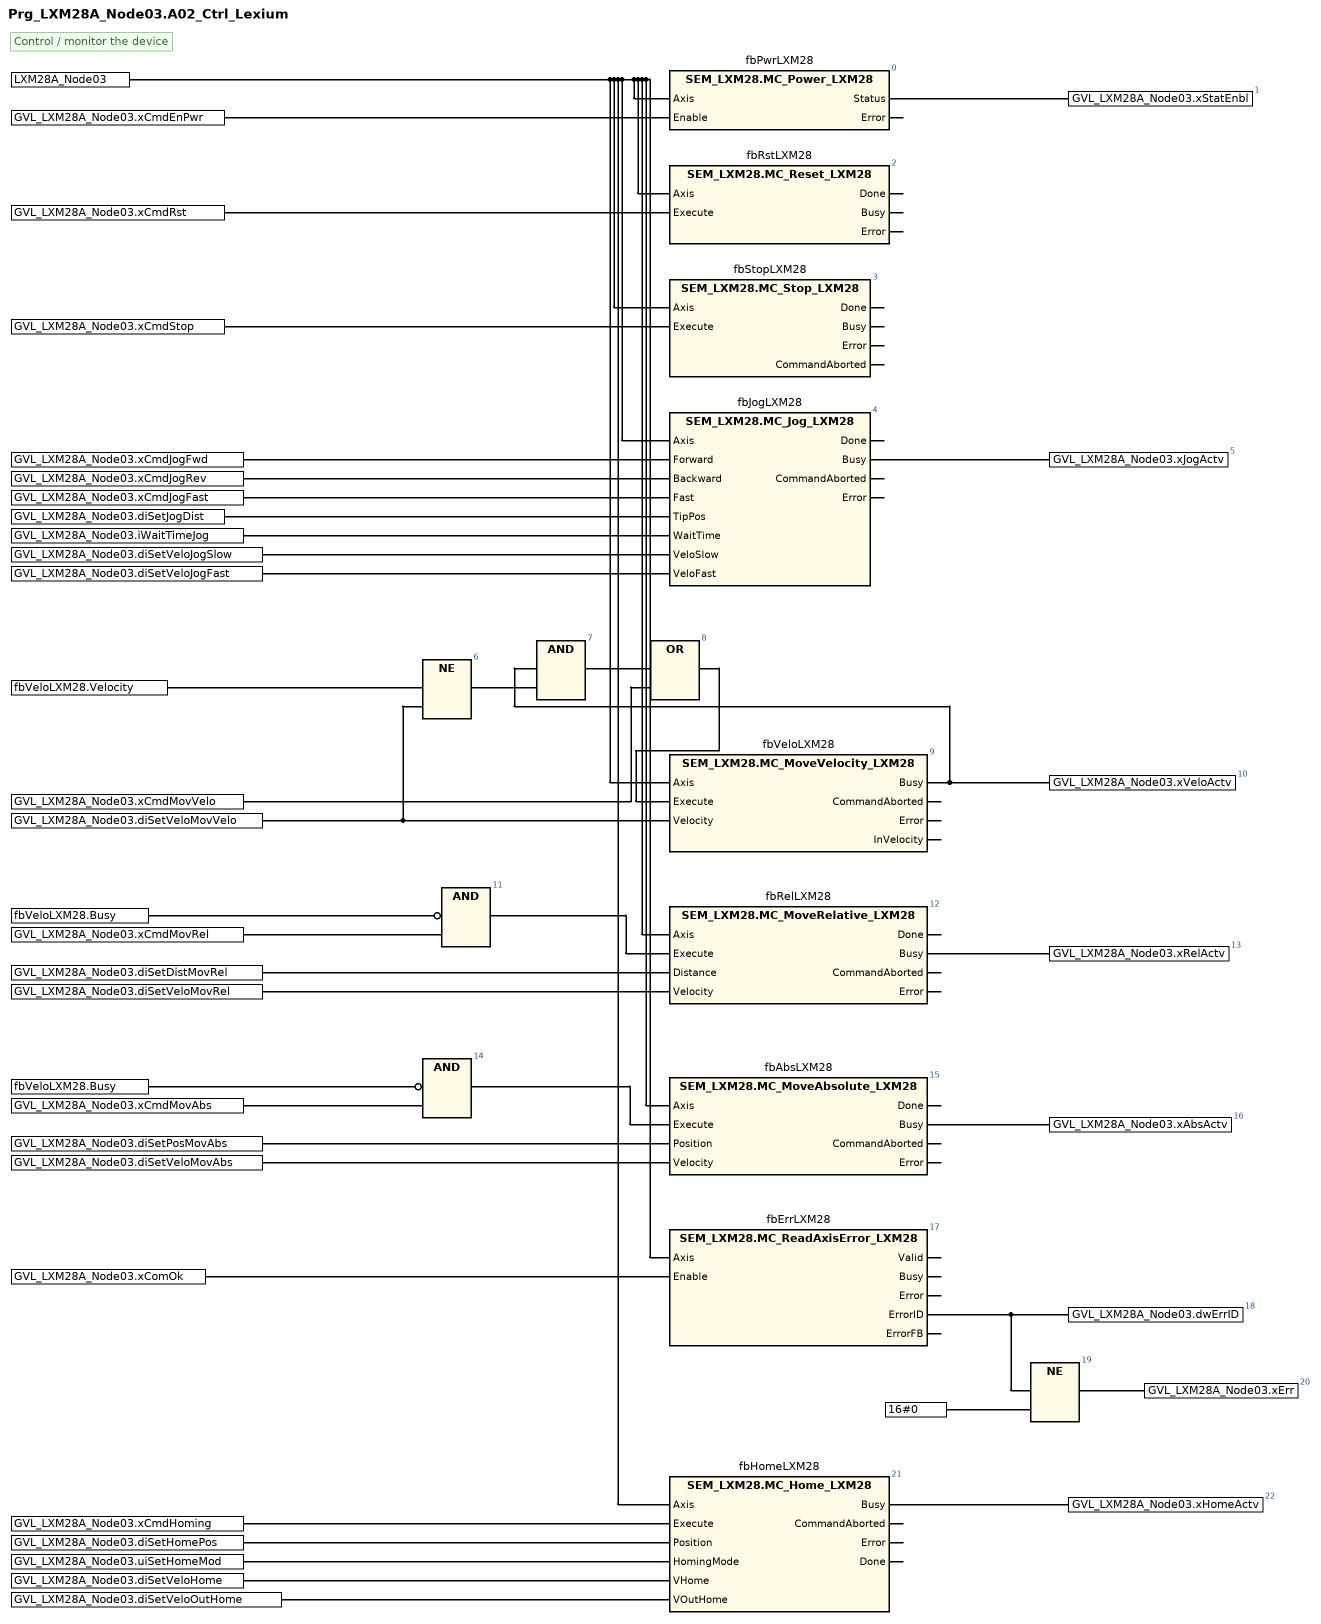
// Control / monitor the device
fbPwrLXM28(Axis := LXM28A_Node03, Enable := GVL_LXM28A_Node03.xCmdEnPwr); // SEM_LXM28.MC_Power_LXM28
GVL_LXM28A_Node03.xStatEnbl := fbPwrLXM28.Status;
fbRstLXM28(Axis := LXM28A_Node03, Execute := GVL_LXM28A_Node03.xCmdRst); // SEM_LXM28.MC_Reset_LXM28
fbStopLXM28(Axis := LXM28A_Node03, Execute := GVL_LXM28A_Node03.xCmdStop); // SEM_LXM28.MC_Stop_LXM28
fbJogLXM28(
    Axis := LXM28A_Node03,
    Forward := GVL_LXM28A_Node03.xCmdJogFwd,
    Backward := GVL_LXM28A_Node03.xCmdJogRev,
    Fast := GVL_LXM28A_Node03.xCmdJogFast,
    TipPos := GVL_LXM28A_Node03.diSetJogDist,
    WaitTime := GVL_LXM28A_Node03.iWaitTimeJog,
    VeloSlow := GVL_LXM28A_Node03.diSetVeloJogSlow,
    VeloFast := GVL_LXM28A_Node03.diSetVeloJogFast); // SEM_LXM28.MC_Jog_LXM28
GVL_LXM28A_Node03.xJogActv := fbJogLXM28.Busy;
fbVeloLXM28(
    Axis := LXM28A_Node03,
    Execute := fbVeloLXM28.Busy AND fbVeloLXM28.Velocity <> GVL_LXM28A_Node03.diSetVeloMovVelo OR GVL_LXM28A_Node03.xCmdMovVelo,
    Velocity := GVL_LXM28A_Node03.diSetVeloMovVelo); // SEM_LXM28.MC_MoveVelocity_LXM28
GVL_LXM28A_Node03.xVeloActv := fbVeloLXM28.Busy;
fbRelLXM28(
    Axis := LXM28A_Node03,
    Execute := NOT fbVeloLXM28.Busy AND GVL_LXM28A_Node03.xCmdMovRel,
    Distance := GVL_LXM28A_Node03.diSetDistMovRel,
    Velocity := GVL_LXM28A_Node03.diSetVeloMovRel); // SEM_LXM28.MC_MoveRelative_LXM28
GVL_LXM28A_Node03.xRelActv := fbRelLXM28.Busy;
fbAbsLXM28(
    Axis := LXM28A_Node03,
    Execute := NOT fbVeloLXM28.Busy AND GVL_LXM28A_Node03.xCmdMovAbs,
    Position := GVL_LXM28A_Node03.diSetPosMovAbs,
    Velocity := GVL_LXM28A_Node03.diSetVeloMovAbs); // SEM_LXM28.MC_MoveAbsolute_LXM28
GVL_LXM28A_Node03.xAbsActv := fbAbsLXM28.Busy;
fbErrLXM28(Axis := LXM28A_Node03, Enable := GVL_LXM28A_Node03.xComOk); // SEM_LXM28.MC_ReadAxisError_LXM28
GVL_LXM28A_Node03.dwErrID := fbErrLXM28.ErrorID;
GVL_LXM28A_Node03.xErr := fbErrLXM28.ErrorID <> 16#0;
fbHomeLXM28(
    Axis := LXM28A_Node03,
    Execute := GVL_LXM28A_Node03.xCmdHoming,
    Position := GVL_LXM28A_Node03.diSetHomePos,
    HomingMode := GVL_LXM28A_Node03.uiSetHomeMod,
    VHome := GVL_LXM28A_Node03.diSetVeloHome,
    VOutHome := GVL_LXM28A_Node03.diSetVeloOutHome); // SEM_LXM28.MC_Home_LXM28
GVL_LXM28A_Node03.xHomeActv := fbHomeLXM28.Busy;
END_ACTION

ACTION A01_GetNodeState:
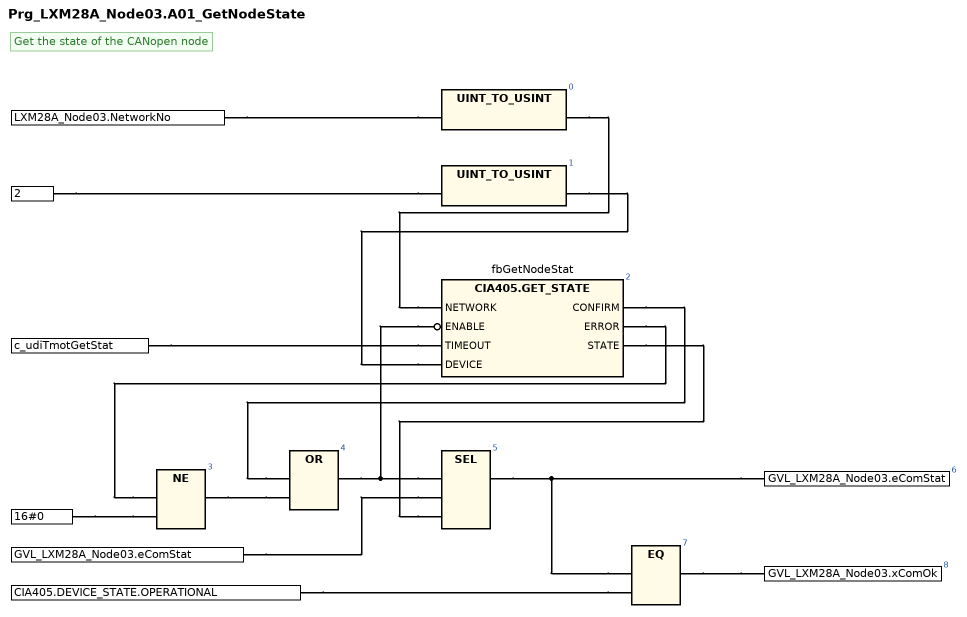
// Get the state of the CANopen node
fbGetNodeStat(
    NETWORK := UINT_TO_USINT(LXM28A_Node03.NetworkNo),
    ENABLE := NOT _w1,
    TIMEOUT := c_udiTmotGetStat,
    DEVICE := UINT_TO_USINT(2)); // CIA405.GET_STATE
_w1 := fbGetNodeStat.CONFIRM OR fbGetNodeStat.ERROR <> 16#0;
_w2 := SEL(_w1, GVL_LXM28A_Node03.eComStat, fbGetNodeStat.STATE);
GVL_LXM28A_Node03.eComStat := _w2;
GVL_LXM28A_Node03.xComOk := _w2 = CIA405.DEVICE_STATE.OPERATIONAL;
END_ACTION

END_PROGRAM

// HMISAC/Application/LXM28A_Node04/Prg_LXM28A_Node04
PROGRAM Prg_LXM28A_Node04
VAR
	fbGetNodeStat     : CIA405.GET_STATE; // FB instance to get the state of the CANopen node
	fbPwrLXM28		  : SEM_LXM28.MC_Power_LXM28; // FB instance to power the Lexium
	fbRstLXM28		  : SEM_LXM28.MC_Reset_LXM28; // FB instance to reset the Lexium
	fbStopLXM28		  : SEM_LXM28.MC_Stop_LXM28; // FB instance to stop the Lexium
	fbJogLXM28		  : SEM_LXM28.MC_Jog_LXM28; // FB instance to turn the drive manually
	fbVeloLXM28	 	  : SEM_LXM28.MC_MoveVelocity_LXM28; // FB instance to start the Lexium in operating mode Profile Velocity
	fbRelLXM28	 	  : SEM_LXM28.MC_MoveRelative_LXM28; // FB instance to start a movement by the defined distance
	fbAbsLXM28	 	  : SEM_LXM28.MC_MoveAbsolute_LXM28; // FB instance to start a movement to the defined absolute target position
	fbErrLXM28	 	  : SEM_LXM28.MC_ReadAxisError_LXM28; // FB instance to read the error state of the Lexium
	fbHomeLXM28	  	  : SEM_LXM28.MC_Home_LXM28; // FB instance to start a reference movement					
END_VAR
VAR CONSTANT
	c_udiTmotGetStat : UDINT := 1000; // Parameter timeout for FB GET_STATE in ms
END_VAR
VAR // added by the converter: edge detectors and wires of the graphical bodies
    _w1, _w2 : ANY;
END_VAR

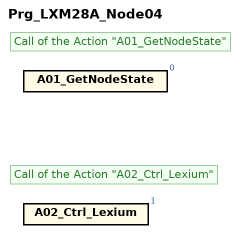
// Call of the Action "A01_GetNodeState"
A01_GetNodeState();
// Call of the Action "A02_Ctrl_Lexium"
A02_Ctrl_Lexium();

ACTION A01_GetNodeState:
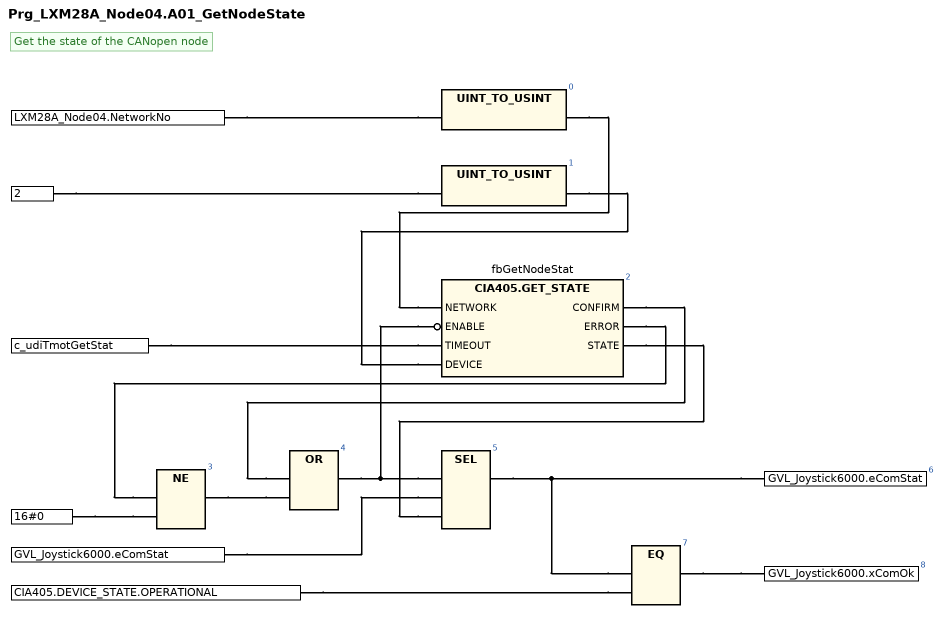
// Get the state of the CANopen node
fbGetNodeStat(
    NETWORK := UINT_TO_USINT(LXM28A_Node04.NetworkNo),
    ENABLE := NOT _w1,
    TIMEOUT := c_udiTmotGetStat,
    DEVICE := UINT_TO_USINT(2)); // CIA405.GET_STATE
_w1 := fbGetNodeStat.CONFIRM OR fbGetNodeStat.ERROR <> 16#0;
_w2 := SEL(_w1, GVL_Joystick6000.eComStat, fbGetNodeStat.STATE);
GVL_Joystick6000.eComStat := _w2;
GVL_Joystick6000.xComOk := _w2 = CIA405.DEVICE_STATE.OPERATIONAL;
END_ACTION

ACTION A02_Ctrl_Lexium:
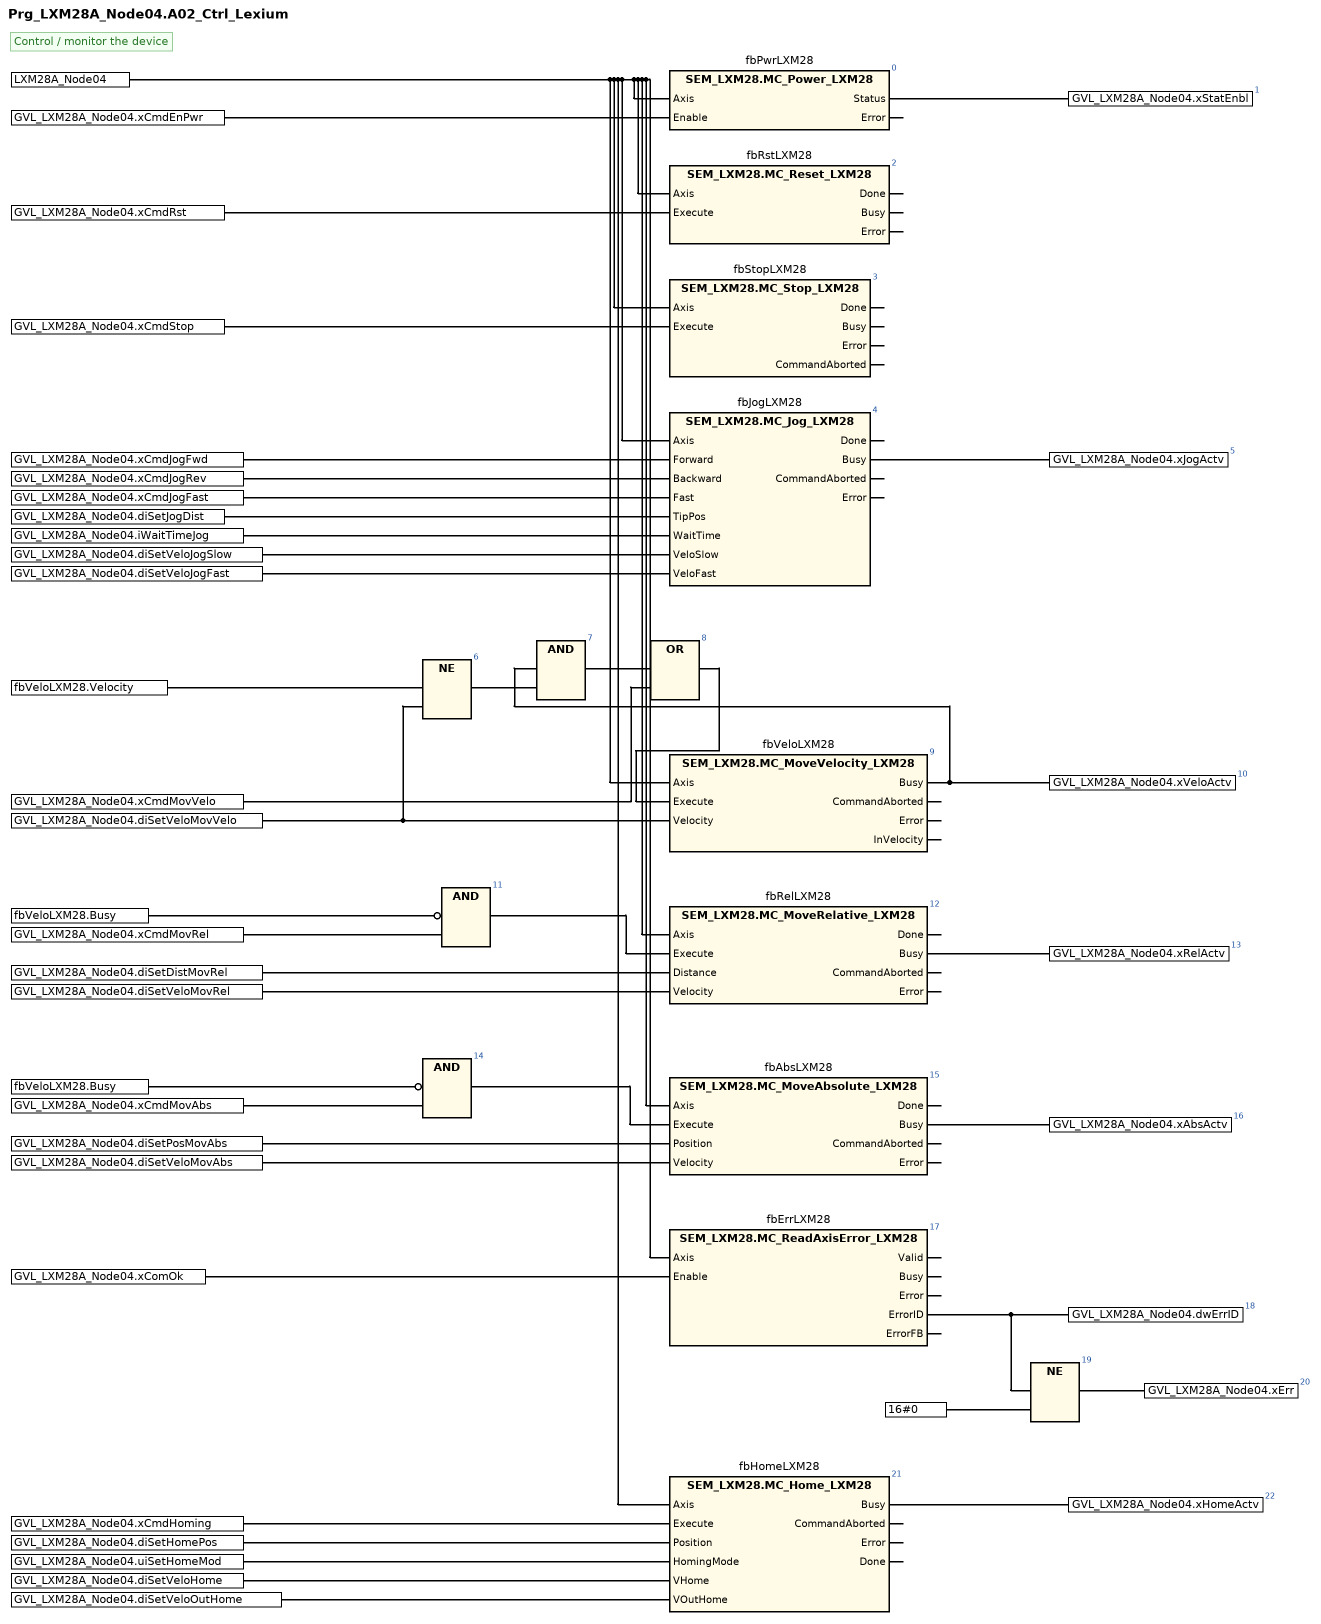
// Control / monitor the device
fbPwrLXM28(Axis := LXM28A_Node04, Enable := GVL_LXM28A_Node04.xCmdEnPwr); // SEM_LXM28.MC_Power_LXM28
GVL_LXM28A_Node04.xStatEnbl := fbPwrLXM28.Status;
fbRstLXM28(Axis := LXM28A_Node04, Execute := GVL_LXM28A_Node04.xCmdRst); // SEM_LXM28.MC_Reset_LXM28
fbStopLXM28(Axis := LXM28A_Node04, Execute := GVL_LXM28A_Node04.xCmdStop); // SEM_LXM28.MC_Stop_LXM28
fbJogLXM28(
    Axis := LXM28A_Node04,
    Forward := GVL_LXM28A_Node04.xCmdJogFwd,
    Backward := GVL_LXM28A_Node04.xCmdJogRev,
    Fast := GVL_LXM28A_Node04.xCmdJogFast,
    TipPos := GVL_LXM28A_Node04.diSetJogDist,
    WaitTime := GVL_LXM28A_Node04.iWaitTimeJog,
    VeloSlow := GVL_LXM28A_Node04.diSetVeloJogSlow,
    VeloFast := GVL_LXM28A_Node04.diSetVeloJogFast); // SEM_LXM28.MC_Jog_LXM28
GVL_LXM28A_Node04.xJogActv := fbJogLXM28.Busy;
fbVeloLXM28(
    Axis := LXM28A_Node04,
    Execute := fbVeloLXM28.Busy AND fbVeloLXM28.Velocity <> GVL_LXM28A_Node04.diSetVeloMovVelo OR GVL_LXM28A_Node04.xCmdMovVelo,
    Velocity := GVL_LXM28A_Node04.diSetVeloMovVelo); // SEM_LXM28.MC_MoveVelocity_LXM28
GVL_LXM28A_Node04.xVeloActv := fbVeloLXM28.Busy;
fbRelLXM28(
    Axis := LXM28A_Node04,
    Execute := NOT fbVeloLXM28.Busy AND GVL_LXM28A_Node04.xCmdMovRel,
    Distance := GVL_LXM28A_Node04.diSetDistMovRel,
    Velocity := GVL_LXM28A_Node04.diSetVeloMovRel); // SEM_LXM28.MC_MoveRelative_LXM28
GVL_LXM28A_Node04.xRelActv := fbRelLXM28.Busy;
fbAbsLXM28(
    Axis := LXM28A_Node04,
    Execute := NOT fbVeloLXM28.Busy AND GVL_LXM28A_Node04.xCmdMovAbs,
    Position := GVL_LXM28A_Node04.diSetPosMovAbs,
    Velocity := GVL_LXM28A_Node04.diSetVeloMovAbs); // SEM_LXM28.MC_MoveAbsolute_LXM28
GVL_LXM28A_Node04.xAbsActv := fbAbsLXM28.Busy;
fbErrLXM28(Axis := LXM28A_Node04, Enable := GVL_LXM28A_Node04.xComOk); // SEM_LXM28.MC_ReadAxisError_LXM28
GVL_LXM28A_Node04.dwErrID := fbErrLXM28.ErrorID;
GVL_LXM28A_Node04.xErr := fbErrLXM28.ErrorID <> 16#0;
fbHomeLXM28(
    Axis := LXM28A_Node04,
    Execute := GVL_LXM28A_Node04.xCmdHoming,
    Position := GVL_LXM28A_Node04.diSetHomePos,
    HomingMode := GVL_LXM28A_Node04.uiSetHomeMod,
    VHome := GVL_LXM28A_Node04.diSetVeloHome,
    VOutHome := GVL_LXM28A_Node04.diSetVeloOutHome); // SEM_LXM28.MC_Home_LXM28
GVL_LXM28A_Node04.xHomeActv := fbHomeLXM28.Busy;
END_ACTION

END_PROGRAM
